INTERFACE I_ArrayDatatype EXTENDS I_UserDefinedDatatype

PROPERTY Dimention : UDINT
GET
END_GET
END_PROPERTY

METHOD TryGetLowerBound : BOOL
VAR_INPUT
	Dimention : UDINT;
	Destination : REFERENCE TO DINT;
END_VAR
END_METHOD

METHOD TryGetUpperBound : BOOL
VAR_INPUT
	Dimention : UDINT;
	Destination : REFERENCE TO DINT;
END_VAR
END_METHOD

METHOD PUBLIC TryResolveAs1DArrayDatatype : BOOL
VAR_INPUT
	Destination : REFERENCE TO I_ArrayDatatype_1D;
END_VAR
END_METHOD

METHOD PUBLIC TryResolveAs2DArrayDatatype : BOOL
VAR_INPUT
	Destination : REFERENCE TO I_ArrayDatatype_2D;
END_VAR
END_METHOD

METHOD PUBLIC TryResolveAs3DArrayDatatype : BOOL
VAR_INPUT
	Destination : REFERENCE TO I_ArrayDatatype_3D;
END_VAR
END_METHOD

END_INTERFACE

(* stored: Version 1.1.0.1, ProductVersion 3.1.4024.13
   Itf I_ArrayDatatype: Id {a8e57a5b-bfda-0173-132d-0647d5e8567e}
   Property Dimention: Id {be1fb109-0ba8-07ed-024c-2305193d98ca}
   Get Get: Id {fe5c673e-18e8-0edc-05c0-f82ce999e57e}
   Method TryGetLowerBound: Id {6864720b-2d0e-07fd-38a5-cca1bb55b3e5}
   Method TryGetUpperBound: Id {b9333345-152f-080b-3047-9d07a376b50b}
   Method TryResolveAs1DArrayDatatype: Id {8dd4a298-7bd3-05ea-21dc-2b952e48cd64}
   Method TryResolveAs2DArrayDatatype: Id {4cca6520-8e58-0fea-39a1-23b7233134f6}
   Method TryResolveAs3DArrayDatatype: Id {f388c645-feb3-0679-314c-0dc086cfc97f} *)
